// TIA Portal V20 export
VAR_GLOBAL   // PLC tag table "Gate1"
   Prox1 AT %I0.0 : Bool;   // Stato sensore prossimità cancello 1 (Aperto -> False)
   Prox2 AT %I0.1 : Bool;   // Stato sensore prossimità cancello 2 (Aperto -> False)
   Prox3 AT %I0.2 : Bool;   // Stato sensore prossimità cancello 3 (Aperto -> False)
END_VAR
